# EPICS autosave request: urRobotApp/Db/waypointJ_settings.req
$(P)$(R)WaypointJ:$(N):Name.VAL
$(P)$(R)WaypointJ:$(N):J1.VAL
$(P)$(R)WaypointJ:$(N):J2.VAL
$(P)$(R)WaypointJ:$(N):J3.VAL
$(P)$(R)WaypointJ:$(N):J4.VAL
$(P)$(R)WaypointJ:$(N):J5.VAL
$(P)$(R)WaypointJ:$(N):J6.VAL
$(P)$(R)WaypointJ:$(N):Gripper.VAL
$(P)$(R)WaypointJ:$(N):Speed.VAL
$(P)$(R)WaypointJ:$(N):Acceleration.VAL
$(P)$(R)WaypointJ:$(N):Blend.VAL
